(* PLC project TestUml.project, Rexroth ctrlX PLC Engineering ctrlX PLC 1.20.12 *)
(* stored: creationDateTime 2025-03-04T16:25:23.2374387, modificationDateTime 2025-03-04T16:13:03.9525114 *)

FUNCTION_BLOCK FB_Count
  VAR_OUTPUT
    iCounter : INT;
  END_VAR

            
          

METHOD M_Count : BOOL
                  iCounter := iCounter + 1;
                
END_METHOD
END_FUNCTION_BLOCK

FUNCTION_BLOCK FB_CountExtended EXTENDS FB_Count
  VAR_OUTPUT
    iExtendedCounter : INT;
  END_VAR

            SUPER^.M_Count();
THIS^.M_Count();
          

METHOD M_Count : BOOL
                  iExtendedCounter := iExtendedCounter - 1;
                
END_METHOD
END_FUNCTION_BLOCK

PROGRAM PRG_Count
  VAR
    fbCountExtended : FB_CountExtended;
    iTestOne : INT;
    iTestTwo : INT;
  END_VAR

            fbCountExtended();

iTestOne := fbCountExtended.iCounter;
iTestTwo := fbCountExtended.iExtendedCounter;
          
END_PROGRAM
